SUBAPPLICATION Uebung_004b_AX (* Toggle Flip-Flop mit IE / E_SWITCH + E_SR *)
  (* Standard: 61499-2; Description: Copyright (c) 2023 Meisterschulen am Ostbahnhof This program and the accompanying materials are made available under the terms of the Eclipse Public License 2.0 which is available at https://www.eclipse.org/legal/epl-2.0/ SPDX-License-Identifier: EPL-2.0 *)
  (* Version 1.0, 2023-10-23, Franz Höpfinger, Meisterschulen am Ostbahnhof, initial API and implementation and/or initial documentation *)
  PACKAGE Uebungen;
  IMPORT logiBUS::io::DI::logiBUS_DI::Input_I1;
  IMPORT logiBUS::io::DI::logiBUS_DI_Events::BUTTON_SINGLE_CLICK;
  IMPORT logiBUS::io::DQ::logiBUS_DO::Output_Q1;
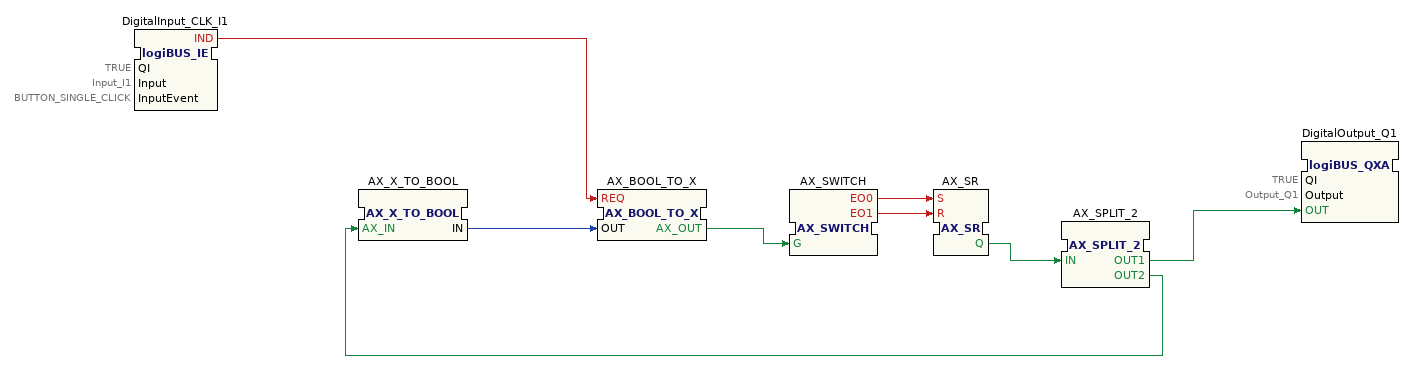
  (* Kommentar FH: nicht empfohlen !!! viel zu viel Bausteine *)
  FBS
    DigitalOutput_Q1 : logiBUS::io::DQ::logiBUS_QXA(QI := TRUE, Output := Output_Q1);
    DigitalInput_CLK_I1 : logiBUS::io::DI::logiBUS_IE(QI := TRUE, Input := Input_I1, InputEvent := BUTTON_SINGLE_CLICK);
    AX_SR : adapter::events::unidirectional::AX_SR;
    AX_SWITCH : adapter::events::unidirectional::AX_SWITCH;
    AX_SPLIT_2 : adapter::events::unidirectional::AX_SPLIT_2;
    AX_BOOL_TO_X : adapter::conversion::unidirectional::AX_BOOL_TO_X;
    AX_X_TO_BOOL : adapter::conversion::unidirectional::AX_X_TO_BOOL;
  END_FBS
  EVENT_CONNECTIONS
    AX_SWITCH.EO0 TO AX_SR.S;
    AX_SWITCH.EO1 TO AX_SR.R;
    DigitalInput_CLK_I1.IND TO AX_BOOL_TO_X.REQ;
  END_CONNECTIONS
  DATA_CONNECTIONS
    AX_X_TO_BOOL.IN TO AX_BOOL_TO_X.OUT;
  END_CONNECTIONS
  ADAPTER_CONNECTIONS
    AX_SR.Q TO AX_SPLIT_2.IN;
    AX_SPLIT_2.OUT1 TO DigitalOutput_Q1.OUT;
    AX_BOOL_TO_X.AX_OUT TO AX_SWITCH.G;
    AX_SPLIT_2.OUT2 TO AX_X_TO_BOOL.AX_IN;
  END_CONNECTIONS
END_SUBAPPLICATION
